// TIA Portal V21 export
// export: Created 2026-07-27T22:11:03.5219089Z, ExportSetting WithDefaults, DisplayName Totally Integrated Automation Portal, DisplayVersion V21, DisplayName SINAMICS Startdrive Advanced, DisplayVersion V21, DisplayName SINAMICS Startdrive G110M, G120, G120C, G120D, G120P, G115D, DisplayVersion V21, DisplayName SINAMICS Startdrive G130, G150, S120, S150, G200, G220, S200, S210, S220, Innomotics MVD, DisplayVersion V21, DisplayName STEP 7 Professional, DisplayVersion V21, DisplayName STEP 7 Safety, DisplayVersion V21, DisplayName Tech WebApplication, DisplayVersion V21, DisplayName WinCC Basic/Comfort/Advanced, DisplayVersion V21, DisplayName WinCC Professional, DisplayVersion V21, DisplayName WinCC Unified, DisplayVersion V21
FUNCTION "PARTIDA_MOTOR_1 (S-01A)" : Void   // FC148, LAD
{ S7_Optimized_Access := 'TRUE' }
VERSION : 0.1
// Network 1: Set memórias entradas digitais
// Network 2: Function Block FALHA
// Network 3: MODO AUTOMÁTICO: Condições para Modo Automático
// Network 4: Alternância/Rotatividade de bombas Principal-Reserva
// Network 5: Function Block CONDIÇÃO DE PARTIDA
// Network 6: Setpoint Manual - Velocidade Proporcial ao Sinal de Saída
// Network 7: Reset Comando Liga
// Network 8: Intertravamento para habilitar o botão liga na IHM
// Network 9: Intertravamento de Segurança
// Network 10: Bloco de Controle Inversor Profinet
// Network 11: Aciona saída digital para partir o motor/bomba
// Network 1: Set memórias entradas digitais
// Network 2: Function Block FALHA
// Network 3: MODO AUTOMÁTICO: Condições para Modo Automático
// Network 4: Alternância/Rotatividade de bombas Principal-Reserva
// Network 5: Function Block CONDIÇÃO DE PARTIDA
// Network 6: Reset Comando Liga
// Network 7: Function Block MODOS DE OPERAÇÃO - Atribuição dos Modos de Operação
// Network 8: Intertravamento para habilitar o botão liga na IHM
// Network 9: Intertravamento de Segurança
// Network 10: Function Block SUCÇÃO OK
// Network 11: Aciona saída digital para partir o motor/bomba
// Network 12: Function Block HORÍMETRO - Tempo de bomba ligada em horas
// stored: AutoNumber true, IsIECCheckEnabled false, SetENOAutomatically false, UDAEnableTagReadback false
   VAR_TEMP   // added for the SCL form of the ladder/FBD networks
      _w1 : Bool;
   END_VAR
BEGIN

REGION Network 1: Set memórias entradas digitais
   // Instanciando entradas digitais em PLC Tags "%M " Address
   // 
   // MODO LOCAL: Indica Operação Local da bomba.
   // MODO REMOTO: Indica Operação Remoto da bomba (IHM).
   // LIGADO: Indica bomba ligada (caso, via sinal discreto).
   // FALHA: Sinal de Falha (caso, via sinal discreto).
   // Instanciando entradas digitais em PLC Tags "M" Address
   // 
   // MODO LOCAL: Indica Operação Local da bomba
   // MODO REMOTO: Indica Operação Remoto da bomba (IHM)
   // LIGADO: Indica bomba ligada
   // FALHA: Sinal de Falha
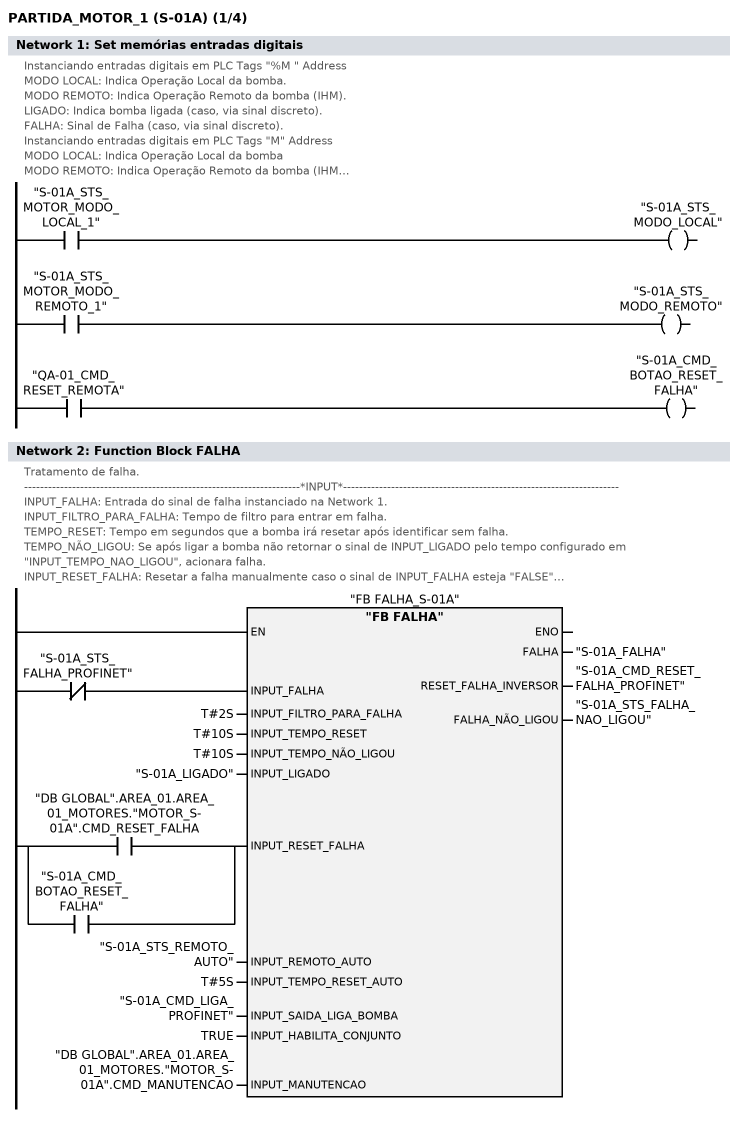
   RUNG wire#powerrail
      Contact( "S-01A_STS_MOTOR_MODO_LOCAL_1" )
      Coil( "S-01A_STS_MODO_LOCAL" )
   END_RUNG
   RUNG wire#powerrail
      Contact( "S-01A_STS_MOTOR_MODO_REMOTO_1" )
      Coil( "S-01A_STS_MODO_REMOTO" )
   END_RUNG
   RUNG wire#powerrail
      Contact( "QA-01_CMD_RESET_REMOTA" )
      Coil( "S-01A_CMD_BOTAO_RESET_FALHA" )
   END_RUNG
   // the same network as SCL:
   "S-01A_STS_MODO_LOCAL" := "S-01A_STS_MOTOR_MODO_LOCAL_1";
   "S-01A_STS_MODO_REMOTO" := "S-01A_STS_MOTOR_MODO_REMOTO_1";
   "S-01A_CMD_BOTAO_RESET_FALHA" := "QA-01_CMD_RESET_REMOTA";
END_REGION

REGION Network 2: Function Block FALHA
   // Tratamento de falha.
   // ---------------------------------------------------------------------*INPUT*---------------------------------------------------------------------
   // INPUT_FALHA: Entrada do sinal de falha instanciado na Network 1.
   // INPUT_FILTRO_PARA_FALHA: Tempo de filtro para entrar em falha.
   // TEMPO_RESET: Tempo em segundos que a bomba irá resetar após identificar sem falha.
   // TEMPO_NÃO_LIGOU: Se após ligar a bomba não retornar o sinal de INPUT_LIGADO pelo tempo configurado em "INPUT_TEMPO_NAO_LIGOU", acionara falha.
   // INPUT_RESET_FALHA: Resetar a falha manualmente caso o sinal de INPUT_FALHA esteja "FALSE".
   // INPUT_REMOTO_AUTO: Caso o equipamento entrar em estado de "FALHA" em "REMOTO_AUTOMATICO" o bloco fará um reset com atraso pelo tempo "INPUT_TEMPO_RESET_AUTO".
   // INPUT_TEMPO_RESET_AUTO: Caso em "REMOTO_AUTO", para resetar será contado o tempo de entrada.
   // INPUT_SAIDA_LIGA_BOMBA: Comando de saída para acionar o equipamento.
   // INPUT_HABILITA_CONJUNTO: Comando para casos de Principal e Reserva (padrão "TRUE").
   // INPUT_MANUTENCAO: Comando de manutenção do equipamento intertrava qualquer acionamento e status de "FALHA".
   // ---------------------------------------------------------------------*OUTPUT*---------------------------------------------------------------------
   // FALHA: Sinal de saída de "FALHA" do equipamento.
   // RESET_FALHA_INVERSOR: Comando enviado para reset do inversor em caso de "FALHA".
   // FALHA_NAO_LIGOU: Caso esteja sendo enviado o comando para "LIGAR" e não receber o feedback de ligado, no tempo de "TEMPO_NÃO_LIGOU", o equiapamento entra em "FALHA".
   // Tratamento de falha da bomba
   // INPUT_FALHA: Entrada do sinal de falha instanciado na Network 1.
   // TEMPO_RESET: Tempo em segundos que a bomba irá resetar após identificar sem falha.
   // TEMPO_NÃO_LIGOU: Se após ligar a bomba não retornar o sinal de LIGADO pelo tempo configurado, acionara falha.
   // INPUT_RESET_FALHA: Resetar a falha manualmente caso o sinal de INPUT_FALHA esteja FALSE
   RUNG wire#powerrail
      "FB FALHA_S-01A"(INPUT_FALHA := wire#w1, INPUT_RESET_FALHA := wire#w2, INPUT_FILTRO_PARA_FALHA := T#2S, INPUT_TEMPO_RESET := T#10S, INPUT_TEMPO_NÃO_LIGOU := T#10S, INPUT_LIGADO := "S-01A_LIGADO", INPUT_REMOTO_AUTO := "S-01A_STS_REMOTO_AUTO", INPUT_TEMPO_RESET_AUTO := T#5S, INPUT_SAIDA_LIGA_BOMBA := "S-01A_CMD_LIGA_PROFINET", INPUT_HABILITA_CONJUNTO := TRUE, INPUT_MANUTENCAO := "DB GLOBAL".AREA_01.AREA_01_MOTORES."MOTOR_S-01A".CMD_MANUTENCAO, FALHA => "S-01A_FALHA", RESET_FALHA_INVERSOR => "S-01A_CMD_RESET_FALHA_PROFINET", FALHA_NÃO_LIGOU => "S-01A_STS_FALHA_NAO_LIGOU")
   END_RUNG
   RUNG wire#powerrail
      I_Contact( "S-01A_STS_FALHA_PROFINET" )
   END_RUNG wire#w1
   RUNG wire#powerrail
      Contact( "DB GLOBAL".AREA_01.AREA_01_MOTORES."MOTOR_S-01A".CMD_RESET_FALHA )
   END_RUNG wire#w2
   RUNG wire#powerrail
      Contact( "S-01A_CMD_BOTAO_RESET_FALHA" )
   END_RUNG wire#w2
   // the same network as SCL:
   "FB FALHA_S-01A"(INPUT_FALHA := NOT "S-01A_STS_FALHA_PROFINET",   // "FB FALHA"
                    INPUT_FILTRO_PARA_FALHA := T#2S,
                    INPUT_TEMPO_RESET := T#10S,
                    INPUT_TEMPO_NÃO_LIGOU := T#10S,
                    INPUT_LIGADO := "S-01A_LIGADO",
                    INPUT_RESET_FALHA := "DB GLOBAL".AREA_01.AREA_01_MOTORES."MOTOR_S-01A".CMD_RESET_FALHA OR "S-01A_CMD_BOTAO_RESET_FALHA",
                    INPUT_REMOTO_AUTO := "S-01A_STS_REMOTO_AUTO",
                    INPUT_TEMPO_RESET_AUTO := T#5S,
                    INPUT_SAIDA_LIGA_BOMBA := "S-01A_CMD_LIGA_PROFINET",
                    INPUT_HABILITA_CONJUNTO := TRUE,
                    INPUT_MANUTENCAO := "DB GLOBAL".AREA_01.AREA_01_MOTORES."MOTOR_S-01A".CMD_MANUTENCAO,
                    FALHA => "S-01A_FALHA",
                    RESET_FALHA_INVERSOR => "S-01A_CMD_RESET_FALHA_PROFINET",
                    FALHA_NÃO_LIGOU => "S-01A_STS_FALHA_NAO_LIGOU");
END_REGION

REGION Network 3: MODO AUTOMÁTICO: Condições para Modo Automático
   // ----------------------------------------------------------------------*INPUT*---------------------------------------------------------------------
   // ---------------------------------------------------------------------*OUTPUT*------------------------------------------------------------------
END_REGION

REGION Network 4: Alternância/Rotatividade de bombas Principal-Reserva
   // ----------------------------------------------------------------------*INPUT*---------------------------------------------------------------------
   // ---------------------------------------------------------------------*OUTPUT*------------------------------------------------------------------
END_REGION

REGION Network 5: Function Block CONDIÇÃO DE PARTIDA
   // Varredura de condicionais para ligar
   // ----------------------------------------------------------------------*INPUT*---------------------------------------------------------------------
   // INPUT_LIGADO: Entrada do sinal de ligado instanciado na Network 1.
   // INPUT_DESLIGADO: Entrada do sinal discreto "DESLIGADO" (caso, feedback via sinal discreto).
   // INPUT_FALHA: Entrada do sinal de falha da saída do bloco na Network 2.
   // INPUT_LOCAL: Entrada do sinal de modo local instanciado na Network 1.
   // INPUT_LOC_AUTO: Entrada do sinal do modo Local Automático
   // INPUT_REMOTO: Entrada do sinal de modo remoto instanciado na Network 1.
   // INPUT_FALHA_PROFNET: Entrada do sinal de Falha na comunicação Profinet.
   // INPUT_HABILITA_AUTO: Entrada do Sinal que habilita o modo Automático.
   // INPUT_CMD_LIGA: Entrada do sinal para acionar o equipamento.
   // CMD_MANUTENÇÃO:Comando de manutenção do equipamento intertrava qualquer acionamento.
   // CMD_MODO_OPERAÇÃO: Seleção do modo de operação do equipamento.
   // CMD_RESET_HORIMETRO: Comando para resetar o contador de Horas Trabalhadas.
   // 
   // 
   // ---------------------------------------------------------------------*OUTPUT*------------------------------------------------------------------
   // LIGA_BOMBA: Se TRUE, as condições estão OK para ligar na Network 11.
   // STATUS_MOTOR: Status de saída; 0 = DESLIGADO; 1 = LIGADO; 2 = FALHA; 3 = MANUTENÇÃO.
   // OUTPUT_REMOTO_AUTO: Saída indica que o motor/bomba está em modo Remoto Automático.
   // OUTPUT_MODO_OPERAÇÃO: Modo de operação local/remoto, manual/automático do equipamento
   // STS_HORIMETRO: Contabilização do tempo do equipamento em operação.
   // RESET_CMD_LIGA: Reset da memória de comando "LIGA" em casos do equipamento estar em modo "REMOTO_AUTOMATICO" ou "FALHA" ou "MANUTENÇÃO".
   // Varredura de condicionais para ligar
   // INPUT_LIGADO: Entrada do sinal de ligado instanciado na Network 1.
   // INPUT_FALHA: Entrada do sinal de falha da saída do bloco na Network 2.
   // INPUT_LOCAL: Entrada do sinal de modo local instanciado na Network 1.
   // INPUT_LOC_AUTO: Entrada do sinal do modo Local Automático
   // INPUT_REMOTO: Entrada do sinal de modo remoto instanciado na Network 1.
   // PARÂMETRO: Parâmetro de monitoramento para ligar e desligar a bomba em automático.
   // PARÂMETRO_LIGA/DESLIGA: Cadastros de programação liga/desliga em relação ao parâmetro.
   // CMD: Comandos recebidos pelo bloco
   // STATUS_MOTOR: Status de saída; 0 = DESLIGADO; 1 = LIGADO; 2 = FALHA; 3 = MANUTENÇÃO.
   // LIGA_BOMBA: Se TRUE, as condições estão OK para ligar na 5.
   // REMOTO_MAN: Saída indica que o motor/bomba está em modo Remoto Manual
   // REMOTO_AUTO: Saída indica que o motor/bomba está em modo Remoto Automático
   // LOCAL_MAN: Saída indica que o motor/bomba está em modo Local Manual
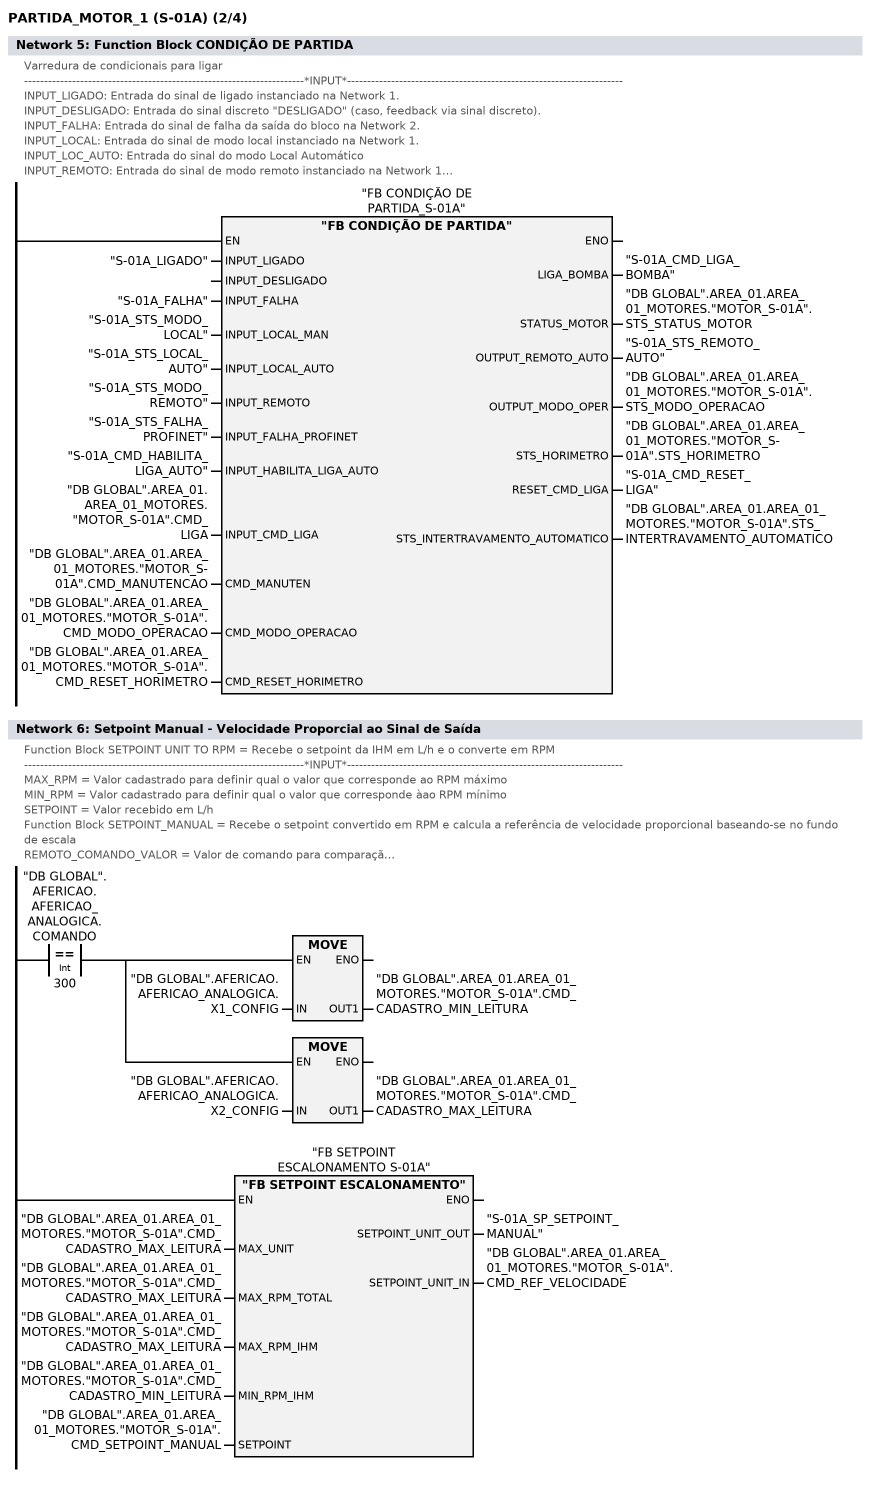
   RUNG wire#powerrail
      "FB CONDIÇÃO DE PARTIDA_S-01A"(INPUT_LIGADO := "S-01A_LIGADO", INPUT_DESLIGADO :=, INPUT_FALHA := "S-01A_FALHA", INPUT_LOCAL_MAN := "S-01A_STS_MODO_LOCAL", INPUT_LOCAL_AUTO := "S-01A_STS_LOCAL_AUTO", INPUT_REMOTO := "S-01A_STS_MODO_REMOTO", INPUT_FALHA_PROFINET := "S-01A_STS_FALHA_PROFINET", INPUT_HABILITA_LIGA_AUTO := "S-01A_CMD_HABILITA_LIGA_AUTO", INPUT_CMD_LIGA := "DB GLOBAL".AREA_01.AREA_01_MOTORES."MOTOR_S-01A".CMD_LIGA, CMD_MANUTEN := "DB GLOBAL".AREA_01.AREA_01_MOTORES."MOTOR_S-01A".CMD_MANUTENCAO, CMD_MODO_OPERACAO := "DB GLOBAL".AREA_01.AREA_01_MOTORES."MOTOR_S-01A".CMD_MODO_OPERACAO, CMD_RESET_HORIMETRO := "DB GLOBAL".AREA_01.AREA_01_MOTORES."MOTOR_S-01A".CMD_RESET_HORIMETRO, LIGA_BOMBA => "S-01A_CMD_LIGA_BOMBA", STATUS_MOTOR => "DB GLOBAL".AREA_01.AREA_01_MOTORES."MOTOR_S-01A".STS_STATUS_MOTOR, OUTPUT_REMOTO_AUTO => "S-01A_STS_REMOTO_AUTO", OUTPUT_MODO_OPER => "DB GLOBAL".AREA_01.AREA_01_MOTORES."MOTOR_S-01A".STS_MODO_OPERACAO, STS_HORIMETRO => "DB GLOBAL".AREA_01.AREA_01_MOTORES."MOTOR_S-01A".STS_HORIMETRO, RESET_CMD_LIGA => "S-01A_CMD_RESET_LIGA", STS_INTERTRAVAMENTO_AUTOMATICO => "DB GLOBAL".AREA_01.AREA_01_MOTORES."MOTOR_S-01A".STS_INTERTRAVAMENTO_AUTOMATICO)
   END_RUNG
   // the same network as SCL:
   "FB CONDIÇÃO DE PARTIDA_S-01A"(INPUT_LIGADO := "S-01A_LIGADO",   // "FB CONDIÇÃO DE PARTIDA"
                           INPUT_FALHA := "S-01A_FALHA",
                           INPUT_LOCAL_MAN := "S-01A_STS_MODO_LOCAL",
                           INPUT_LOCAL_AUTO := "S-01A_STS_LOCAL_AUTO",
                           INPUT_REMOTO := "S-01A_STS_MODO_REMOTO",
                           INPUT_FALHA_PROFINET := "S-01A_STS_FALHA_PROFINET",
                           INPUT_HABILITA_LIGA_AUTO := "S-01A_CMD_HABILITA_LIGA_AUTO",
                           INPUT_CMD_LIGA := "DB GLOBAL".AREA_01.AREA_01_MOTORES."MOTOR_S-01A".CMD_LIGA,
                           CMD_MANUTEN := "DB GLOBAL".AREA_01.AREA_01_MOTORES."MOTOR_S-01A".CMD_MANUTENCAO,
                           CMD_MODO_OPERACAO := "DB GLOBAL".AREA_01.AREA_01_MOTORES."MOTOR_S-01A".CMD_MODO_OPERACAO,
                           CMD_RESET_HORIMETRO := "DB GLOBAL".AREA_01.AREA_01_MOTORES."MOTOR_S-01A".CMD_RESET_HORIMETRO,
                           LIGA_BOMBA => "S-01A_CMD_LIGA_BOMBA",
                           STATUS_MOTOR => "DB GLOBAL".AREA_01.AREA_01_MOTORES."MOTOR_S-01A".STS_STATUS_MOTOR,
                           OUTPUT_REMOTO_AUTO => "S-01A_STS_REMOTO_AUTO",
                           OUTPUT_MODO_OPER => "DB GLOBAL".AREA_01.AREA_01_MOTORES."MOTOR_S-01A".STS_MODO_OPERACAO,
                           STS_HORIMETRO => "DB GLOBAL".AREA_01.AREA_01_MOTORES."MOTOR_S-01A".STS_HORIMETRO,
                           RESET_CMD_LIGA => "S-01A_CMD_RESET_LIGA",
                           STS_INTERTRAVAMENTO_AUTOMATICO => "DB GLOBAL".AREA_01.AREA_01_MOTORES."MOTOR_S-01A".STS_INTERTRAVAMENTO_AUTOMATICO);
END_REGION

REGION Network 6: Setpoint Manual - Velocidade Proporcial ao Sinal de Saída
   // Function Block SETPOINT UNIT TO RPM = Recebe o setpoint da IHM em L/h e o converte em RPM
   // ----------------------------------------------------------------------*INPUT*---------------------------------------------------------------------
   // MAX_RPM = Valor cadastrado para definir qual o valor que corresponde ao RPM máximo
   // MIN_RPM = Valor cadastrado para definir qual o valor que corresponde àao RPM mínimo
   // SETPOINT = Valor recebido em L/h
   // 
   // Function Block SETPOINT_MANUAL = Recebe o setpoint convertido em RPM e calcula a referência de velocidade proporcional baseando-se no fundo de escala
   // REMOTO_COMANDO_VALOR = Valor de comando para comparação
   // COMANDO = Comando recebido para confirmar setpoint
   // RANGE_MAX: Valor cadastrado para definir qual o valor que corresponde ao RPM máximo
   // RANGE_MIN: Valor cadastrado para definir qual o valor que corresponde àao RPM mínimo
   // VALOR_SAIDA: Valor do setpoint interpretado dentro da escala do CLP correspondente ao sinal elétrico (4-20mA ou 0-10V) que o inversor recebe e ajusta sua saída proporcionalmente.
   // 
   // ---------------------------------------------------------------------*OUTPUT*------------------------------------------------------------------
   RUNG wire#powerrail
      { S7_Templates := "SrcType := Int" } EQ_Contact(in1 := "DB GLOBAL".AFERICAO.AFERICAO_ANALOGICA.COMANDO, in2 := 300)
      wire#w1
      Move(in := "DB GLOBAL".AFERICAO.AFERICAO_ANALOGICA.X1_CONFIG, out1 => "DB GLOBAL".AREA_01.AREA_01_MOTORES."MOTOR_S-01A".CMD_CADASTRO_MIN_LEITURA)
   END_RUNG
   RUNG wire#w1
      Move(in := "DB GLOBAL".AFERICAO.AFERICAO_ANALOGICA.X2_CONFIG, out1 => "DB GLOBAL".AREA_01.AREA_01_MOTORES."MOTOR_S-01A".CMD_CADASTRO_MAX_LEITURA)
   END_RUNG
   RUNG wire#powerrail
      "FB SETPOINT ESCALONAMENTO S-01A"(MAX_UNIT := "DB GLOBAL".AREA_01.AREA_01_MOTORES."MOTOR_S-01A".CMD_CADASTRO_MAX_LEITURA, MAX_RPM_TOTAL := "DB GLOBAL".AREA_01.AREA_01_MOTORES."MOTOR_S-01A".CMD_CADASTRO_MAX_LEITURA, MAX_RPM_IHM := "DB GLOBAL".AREA_01.AREA_01_MOTORES."MOTOR_S-01A".CMD_CADASTRO_MAX_LEITURA, MIN_RPM_IHM := "DB GLOBAL".AREA_01.AREA_01_MOTORES."MOTOR_S-01A".CMD_CADASTRO_MIN_LEITURA, SETPOINT := "DB GLOBAL".AREA_01.AREA_01_MOTORES."MOTOR_S-01A".CMD_SETPOINT_MANUAL, SETPOINT_UNIT_OUT => "S-01A_SP_SETPOINT_MANUAL", SETPOINT_UNIT_IN => "DB GLOBAL".AREA_01.AREA_01_MOTORES."MOTOR_S-01A".CMD_REF_VELOCIDADE)
   END_RUNG
   // the same network as SCL:
   IF "DB GLOBAL".AFERICAO.AFERICAO_ANALOGICA.COMANDO = 300 THEN
       "DB GLOBAL".AREA_01.AREA_01_MOTORES."MOTOR_S-01A".CMD_CADASTRO_MIN_LEITURA := "DB GLOBAL".AFERICAO.AFERICAO_ANALOGICA.X1_CONFIG;
       "DB GLOBAL".AREA_01.AREA_01_MOTORES."MOTOR_S-01A".CMD_CADASTRO_MAX_LEITURA := "DB GLOBAL".AFERICAO.AFERICAO_ANALOGICA.X2_CONFIG;
   END_IF;
   "FB SETPOINT ESCALONAMENTO S-01A"(MAX_UNIT := "DB GLOBAL".AREA_01.AREA_01_MOTORES."MOTOR_S-01A".CMD_CADASTRO_MAX_LEITURA,   // "FB SETPOINT ESCALONAMENTO"
                           MAX_RPM_TOTAL := "DB GLOBAL".AREA_01.AREA_01_MOTORES."MOTOR_S-01A".CMD_CADASTRO_MAX_LEITURA,
                           MAX_RPM_IHM := "DB GLOBAL".AREA_01.AREA_01_MOTORES."MOTOR_S-01A".CMD_CADASTRO_MAX_LEITURA,
                           MIN_RPM_IHM := "DB GLOBAL".AREA_01.AREA_01_MOTORES."MOTOR_S-01A".CMD_CADASTRO_MIN_LEITURA,
                           SETPOINT := "DB GLOBAL".AREA_01.AREA_01_MOTORES."MOTOR_S-01A".CMD_SETPOINT_MANUAL,
                           SETPOINT_UNIT_OUT => "S-01A_SP_SETPOINT_MANUAL",
                           SETPOINT_UNIT_IN => "DB GLOBAL".AREA_01.AREA_01_MOTORES."MOTOR_S-01A".CMD_REF_VELOCIDADE);
END_REGION

REGION Network 7: Reset Comando Liga
   // Condições para resetar o comando liga enviado ao function block CONDIÇÃO DE PARTIDA:
   // Caso o Modo Automático, Falha no motor/bomba ou Modo Manutenção sejam acionados, o Comando Liga será resetado, desligando o motor/bomba.
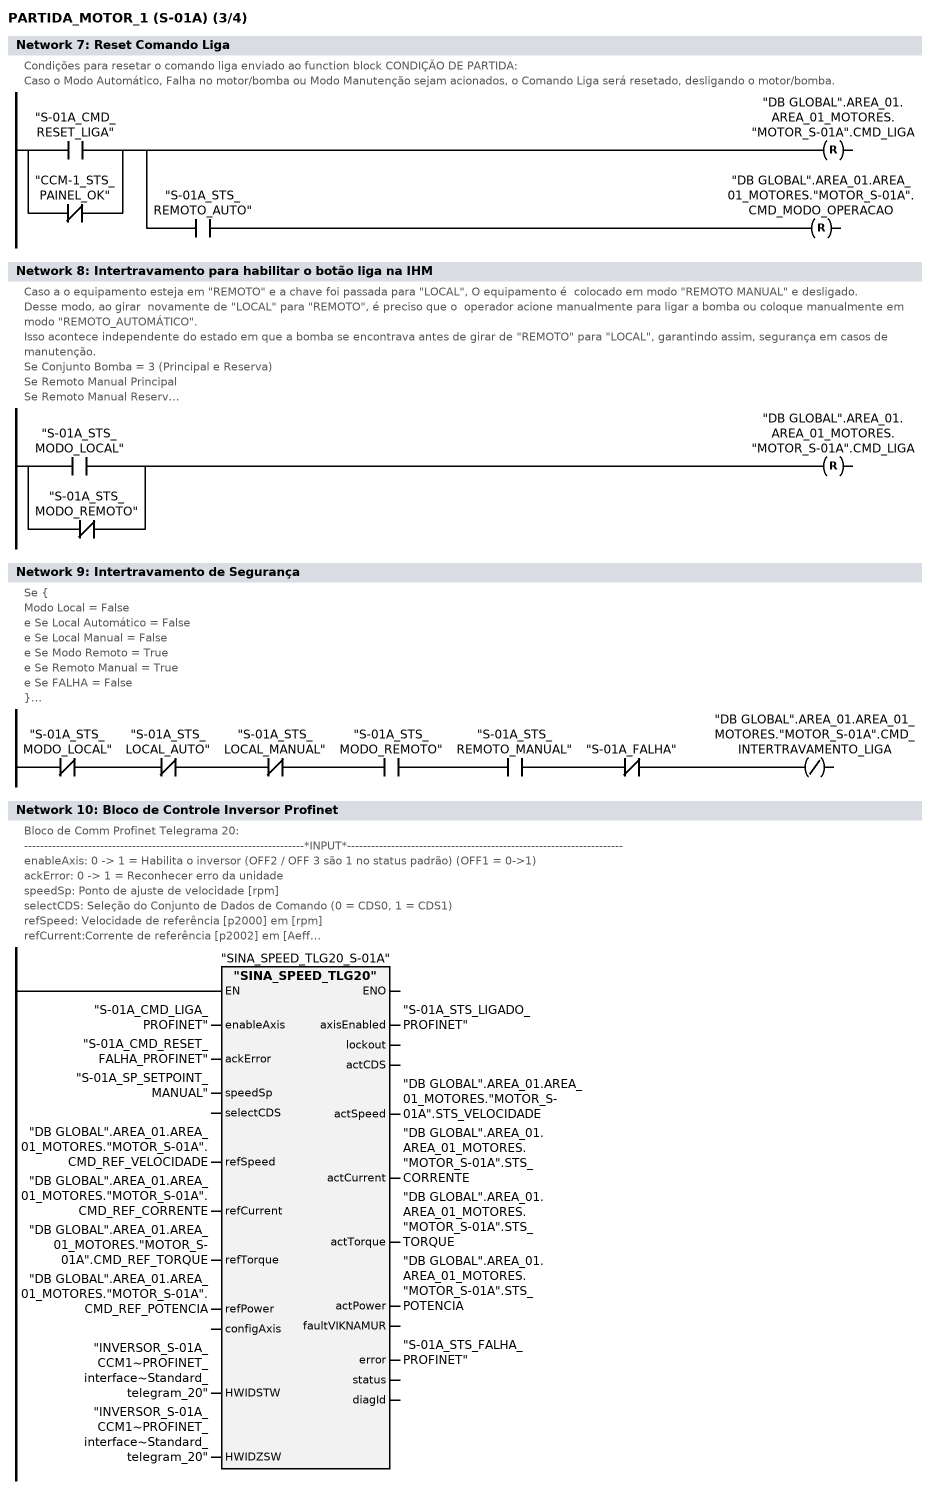
   RUNG wire#powerrail
      Contact( "S-01A_CMD_RESET_LIGA" )
      wire#w1
      R_Coil( "DB GLOBAL".AREA_01.AREA_01_MOTORES."MOTOR_S-01A".CMD_LIGA )
   END_RUNG
   RUNG wire#powerrail
      I_Contact( "CCM-1_STS_PAINEL_OK" )
   END_RUNG wire#w1
   RUNG wire#w1
      Contact( "S-01A_STS_REMOTO_AUTO" )
      R_Coil( "DB GLOBAL".AREA_01.AREA_01_MOTORES."MOTOR_S-01A".CMD_MODO_OPERACAO )
   END_RUNG
   // the same network as SCL:
   #_w1 := "S-01A_CMD_RESET_LIGA" OR NOT "CCM-1_STS_PAINEL_OK";
   IF #_w1 THEN "DB GLOBAL".AREA_01.AREA_01_MOTORES."MOTOR_S-01A".CMD_LIGA := FALSE; END_IF;
   IF #_w1 AND "S-01A_STS_REMOTO_AUTO" THEN
       "DB GLOBAL".AREA_01.AREA_01_MOTORES."MOTOR_S-01A".CMD_MODO_OPERACAO := FALSE;
   END_IF;
END_REGION

REGION Network 8: Intertravamento para habilitar o botão liga na IHM
   // Caso a o equipamento esteja em "REMOTO" e a chave foi passada para "LOCAL", O equipamento é  colocado em modo "REMOTO MANUAL" e desligado.
   // Desse modo, ao girar  novamente de "LOCAL" para "REMOTO", é preciso que o  operador acione manualmente para ligar a bomba ou coloque manualmente em modo "REMOTO_AUTOMÁTICO".
   // Isso acontece independente do estado em que a bomba se encontrava antes de girar de "REMOTO" para "LOCAL", garantindo assim, segurança em casos de manutenção.
   // Se Conjunto Bomba = 3 (Principal e Reserva)
   // Se Remoto Manual Principal
   // Se Remoto Manual Reserva
   // Se Habilitado Liga Principal
   // Se Habilitado Liga Reserva
   // Então Habilita Conjunto de Bomba
   // 
   // Se Conjunto Bomba <> 3
   // Se Remoto Manual Principal
   // Se Habilita Principal 
   // ou
   // Se Remoto Manual Reserva 
   // Se Habilita Reserva
   // Então Habilita Bomba Unitária
   // 
   // Se Bomba Unitária Habilitado
   // ou
   // Se Conjunto Bomba Habilitado
   // Então 
   // Habilita Intertravamento Botão IHM de Conjunto Bomba
   RUNG wire#powerrail
      Contact( "S-01A_STS_MODO_LOCAL" )
      wire#w1
      R_Coil( "DB GLOBAL".AREA_01.AREA_01_MOTORES."MOTOR_S-01A".CMD_LIGA )
   END_RUNG
   RUNG wire#powerrail
      I_Contact( "S-01A_STS_MODO_REMOTO" )
   END_RUNG wire#w1
   // the same network as SCL:
   IF "S-01A_STS_MODO_LOCAL" OR NOT "S-01A_STS_MODO_REMOTO" THEN
       "DB GLOBAL".AREA_01.AREA_01_MOTORES."MOTOR_S-01A".CMD_LIGA := FALSE;
   END_IF;
END_REGION

REGION Network 9: Intertravamento de Segurança
   // Se {
   // Modo Local = False
   // e Se Local Automático = False
   // e Se Local Manual = False
   // e Se Modo Remoto = True
   // e Se Remoto Manual = True
   // e Se FALHA = False
   // } 
   // Habilita botão para ligar manualmente pela IHM.
   // Caso a bomba esteja em REMOTO e a chave foi passada para LOCAL, A bomba é  colocada em modo REMOTO MANUAL E desligada. Desse modo, ao girar  novamente de LOCAL para REMOTO, é preciso que o  operador acione manualmente para ligar a bomba ou coloque manualmente em modo REMOTO AUTOMÁTICO. Isso acontece independente do estado em que a bomba se encontrava antes de girar de REMOTO para LOCAL, garantindo assim, segurança em casos de manutenção.
   RUNG wire#powerrail
      I_Contact( "S-01A_STS_MODO_LOCAL" )
      I_Contact( "S-01A_STS_LOCAL_AUTO" )
      I_Contact( "S-01A_STS_LOCAL_MANUAL" )
      Contact( "S-01A_STS_MODO_REMOTO" )
      Contact( "S-01A_STS_REMOTO_MANUAL" )
      I_Contact( "S-01A_FALHA" )
      I_Coil( "DB GLOBAL".AREA_01.AREA_01_MOTORES."MOTOR_S-01A".CMD_INTERTRAVAMENTO_LIGA )
   END_RUNG
   // the same network as SCL:
   "DB GLOBAL".AREA_01.AREA_01_MOTORES."MOTOR_S-01A".CMD_INTERTRAVAMENTO_LIGA := NOT (NOT "S-01A_STS_MODO_LOCAL" AND NOT "S-01A_STS_LOCAL_AUTO" AND NOT "S-01A_STS_LOCAL_MANUAL" AND "S-01A_STS_MODO_REMOTO" AND "S-01A_STS_REMOTO_MANUAL" AND NOT "S-01A_FALHA");
END_REGION

REGION Network 10: Bloco de Controle Inversor Profinet
   // Bloco de Comm Profinet Telegrama 20:
   // ----------------------------------------------------------------------*INPUT*---------------------------------------------------------------------
   // enableAxis: 0 -> 1 = Habilita o inversor (OFF2 / OFF 3 são 1 no status padrão) (OFF1 = 0->1)
   // ackError: 0 -> 1 = Reconhecer erro da unidade
   // speedSp: Ponto de ajuste de velocidade [rpm]
   // selectCDS: Seleção do Conjunto de Dados de Comando (0 = CDS0, 1 = CDS1)
   // refSpeed: Velocidade de referência [p2000] em [rpm]
   // refCurrent:Corrente de referência [p2002] em [Aeff]
   // refTorque: Torque de referência [p2003] em [Nm]
   // refPower: Potência de referência [r2005] em [kW]
   // configAxis: Entrada binária programada para controlar todas as funções do telegrama sem sua própria entrada de bloco de função
   // HWIDSTW: Slot de ponto de ajuste do identificador de hardware
   // HWIDZSW: Slot de valor real do identificador de hardware
   // ---------------------------------------------------------------------*OUTPUT*------------------------------------------------------------------
   // axisEnabled: 1 = O inversor está habilitado
   // lockout: 1 = Bloqueio do inversor ativo
   // actCDS: Conjunto de dados de comando ativo (0 = CDS0, 1 = CDS1)
   // actSpeed: Velocidade real suavizada em [1/min]
   // actCurrent: Corrente real suavizada em [Arms]
   // actTorque: Torque real suavizado em [Nm]
   // actPower: Potência ativa real suavizada em [kW]
   // faultVIKNAMUR: Palavra de falha de acordo com a definição VIK-NAMUR
   // error: 1 = Erro (FB e Infeed)
   // status: Saída de status (7002 = FB em operação; 7xxx = aviso; 8xxx = descrição do erro - leia o manual)
   // diagId: Códigos de erro dos blocos funcionais do sistema DPWR / DPRD_DAT
   RUNG wire#powerrail
      "SINA_SPEED_TLG20_S-01A"(enableAxis := "S-01A_CMD_LIGA_PROFINET", ackError := "S-01A_CMD_RESET_FALHA_PROFINET", speedSp := "S-01A_SP_SETPOINT_MANUAL", selectCDS :=, refSpeed := "DB GLOBAL".AREA_01.AREA_01_MOTORES."MOTOR_S-01A".CMD_REF_VELOCIDADE, refCurrent := "DB GLOBAL".AREA_01.AREA_01_MOTORES."MOTOR_S-01A".CMD_REF_CORRENTE, refTorque := "DB GLOBAL".AREA_01.AREA_01_MOTORES."MOTOR_S-01A".CMD_REF_TORQUE, refPower := "DB GLOBAL".AREA_01.AREA_01_MOTORES."MOTOR_S-01A".CMD_REF_POTENCIA, configAxis :=, HWIDSTW := "INVERSOR_S-01A_CCM1~PROFINET_interface~Standard_telegram_20", HWIDZSW := "INVERSOR_S-01A_CCM1~PROFINET_interface~Standard_telegram_20", axisEnabled => "S-01A_STS_LIGADO_PROFINET", lockout =>, actCDS =>, actSpeed => "DB GLOBAL".AREA_01.AREA_01_MOTORES."MOTOR_S-01A".STS_VELOCIDADE, actCurrent => "DB GLOBAL".AREA_01.AREA_01_MOTORES."MOTOR_S-01A".STS_CORRENTE, actTorque => "DB GLOBAL".AREA_01.AREA_01_MOTORES."MOTOR_S-01A".STS_TORQUE, actPower => "DB GLOBAL".AREA_01.AREA_01_MOTORES."MOTOR_S-01A".STS_POTENCIA, faultVIKNAMUR =>, error => "S-01A_STS_FALHA_PROFINET", status =>, diagId =>)
   END_RUNG
   // the same network as SCL:
   "SINA_SPEED_TLG20_S-01A"(enableAxis := "S-01A_CMD_LIGA_PROFINET",   // "SINA_SPEED_TLG20"
                           ackError := "S-01A_CMD_RESET_FALHA_PROFINET",
                           speedSp := "S-01A_SP_SETPOINT_MANUAL",
                           refSpeed := "DB GLOBAL".AREA_01.AREA_01_MOTORES."MOTOR_S-01A".CMD_REF_VELOCIDADE,
                           refCurrent := "DB GLOBAL".AREA_01.AREA_01_MOTORES."MOTOR_S-01A".CMD_REF_CORRENTE,
                           refTorque := "DB GLOBAL".AREA_01.AREA_01_MOTORES."MOTOR_S-01A".CMD_REF_TORQUE,
                           refPower := "DB GLOBAL".AREA_01.AREA_01_MOTORES."MOTOR_S-01A".CMD_REF_POTENCIA,
                           HWIDSTW := "INVERSOR_S-01A_CCM1~PROFINET_interface~Standard_telegram_20",
                           HWIDZSW := "INVERSOR_S-01A_CCM1~PROFINET_interface~Standard_telegram_20",
                           axisEnabled => "S-01A_STS_LIGADO_PROFINET",
                           actSpeed => "DB GLOBAL".AREA_01.AREA_01_MOTORES."MOTOR_S-01A".STS_VELOCIDADE,
                           actCurrent => "DB GLOBAL".AREA_01.AREA_01_MOTORES."MOTOR_S-01A".STS_CORRENTE,
                           actTorque => "DB GLOBAL".AREA_01.AREA_01_MOTORES."MOTOR_S-01A".STS_TORQUE,
                           actPower => "DB GLOBAL".AREA_01.AREA_01_MOTORES."MOTOR_S-01A".STS_POTENCIA,
                           error => "S-01A_STS_FALHA_PROFINET");
END_REGION

REGION Network 11: Aciona saída digital para partir o motor/bomba
   // LIGA_BOMBA: Comando recebido pelo bloco FB CONDIÇÃO DE PARTIDA para ligar.
   // SUCÇÂO_OK: Se TRUE, bomba está habilitada para ligar.
   // 
   // Saída digital do CLP que envia o comando de liga para a bomba.
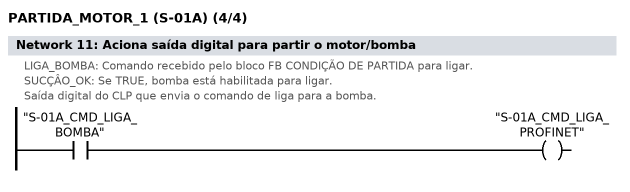
   RUNG wire#powerrail
      Contact( "S-01A_CMD_LIGA_BOMBA" )
      Coil( "S-01A_CMD_LIGA_PROFINET" )
   END_RUNG
   // the same network as SCL:
   "S-01A_CMD_LIGA_PROFINET" := "S-01A_CMD_LIGA_BOMBA";
END_REGION
END_FUNCTION
